// TIA Portal V17 export
// export: Created 2024-03-30T11:15:26.1846062Z, ExportSetting WithDefaults, DisplayName Totally Integrated Automation Portal, DisplayVersion V17, DisplayName TIA Portal Openness, DisplayVersion V17, DisplayName TIA Portal Version Control Interface, DisplayVersion V17, DisplayName STEP 7 Professional, DisplayVersion V17, DisplayName STEP 7 Safety, DisplayVersion V17, DisplayName WinCC Advanced, DisplayVersion V17
TYPE "typ_MQTT_Interface_TXT_Controler_Subscribe"
// stored: IsFailsafeCompliant false
   STRUCT
      State_NFC_Device { S7_SetPoint := 'True'} : "typ_SPS_NFC_Module_State";
   END_STRUCT;
END_TYPE
